PROGRAM ControlQ_LD
VAR
    QueueSTFBD_0 : QueueSTFBD;
    mxQueue : BOOL;
    miOrderQueue : INT;
    Queue : ARRAY [1..3] OF INT;
    ButtonRequstFBD_0 : ButtonRequstFBD;
	QueueSTFBD_2: QueueSTFBD;
	QueueSTFBD_1: QueueSTFBD;
END_VAR
VAR_INPUT
    ixDequeue : BOOL;
    iiOrderDequeue : INT;
END_VAR

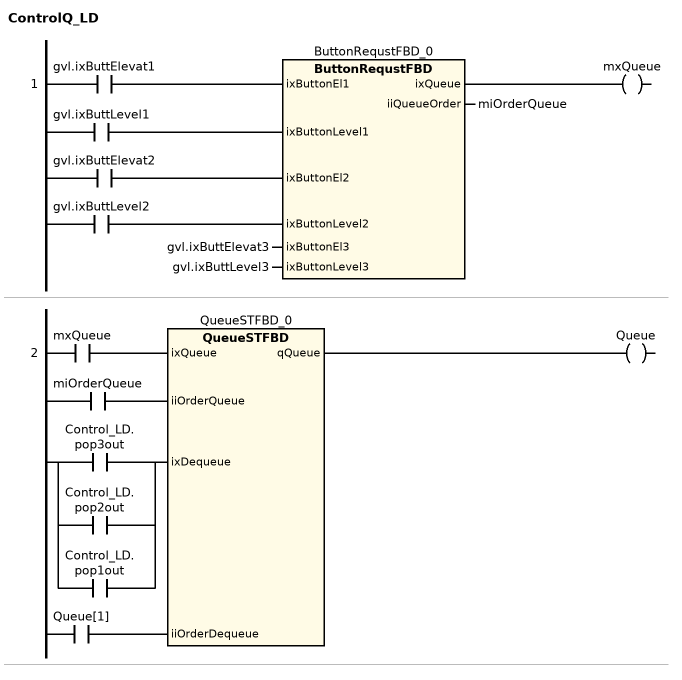
// NETWORK 1
ButtonRequstFBD_0(
    ixButtonEl1 := gvl.ixButtElevat1,
    ixButtonLevel1 := gvl.ixButtLevel1,
    ixButtonEl2 := gvl.ixButtElevat2,
    ixButtonLevel2 := gvl.ixButtLevel2,
    ixButtonEl3 := gvl.ixButtElevat3,
    ixButtonLevel3 := gvl.ixButtLevel3,
    iiQueueOrder => miOrderQueue); // ButtonRequstFBD
mxQueue := ButtonRequstFBD_0.ixQueue;

// NETWORK 2
QueueSTFBD_0(
    ixQueue := mxQueue,
    iiOrderQueue := miOrderQueue,
    ixDequeue := Control_LD.pop3out OR Control_LD.pop2out OR Control_LD.pop1out,
    iiOrderDequeue := Queue[1]); // QueueSTFBD
Queue := QueueSTFBD_0.qQueue;

END_PROGRAM

(* stored: Version 1.1.0.1, ProductVersion 3.1.4024.12
   POU ControlQ_LD: Id {39745b50-a360-41e8-aec4-fabf65da8cf2}, SpecialFunc None *)
